INTERFACE I_ContainTracePublisher EXTENDS I_Base

PROPERTY Publisher : I_TracePublisher
GET
END_GET
END_PROPERTY

END_INTERFACE

(* stored: Version 1.1.0.1, ProductVersion 3.1.4026.18
   Itf I_ContainTracePublisher: Id {18bdaa49-96a9-4979-88e4-db28d5812809}
   Property Publisher: Id {5ec0901d-ee31-4496-acb4-70b44f6d96a8}
   Get Get: Id {74688138-b729-4f3c-b902-bff02adb75b1} *)
